CASE _inst_intStep OF
	0: // Reset FB and set default values
		IF NOT bModbusBusy AND NOT THIS^.P_bError THEN
			IF _in_bValue = TRUE THEN
				fbMBWriteSingleCoil.nValue := 16#FF00;
			ELSE
				fbMBWriteSingleCoil.nValue := 16#0000;
			END_IF
			fbMBWriteSingleCoil(
				sIPAddr:= in_sIPAddr, 
				nTCPPort:= in_uintTCPPort, 
				nUnitID:= in_byteUnitID, 
				nMBAddr:= _in_wordMBAddr, 
				bExecute:= FALSE, 
				tTimeout:= _in_timeTimeout);
		
			THIS^.M_LogMessage('Writing Single Coil');			
			_inst_intStep := 10;
		END_IF
		
		
	10: //Call ReadCoils Beckhoff Action and run it to completion
		fbMBWriteSingleCoil(bExecute := TRUE);
		IF NOT fbMBWriteSingleCoil.bBusy THEN
			fbMBWriteSingleCoil(bExecute:= FALSE);
			_inst_intStep := 20;
		END_IF
		
	20: //If no error, reset steps, else go to error step
		IF NOT fbMBWriteSingleCoil.bError THEN
			M_WriteSingleCoil := TRUE;
			THIS^.M_LogMessage('Write Single Coil Complete');
			_inst_intStep := 0;
		ELSE
			_inst_intStep := 100;
		END_IF
		
	100: //Error
		THIS^.M_SetError(fbMBWriteSingleCoil.nErrId,
							'Error occurred when writing single coil.');
		_inst_intStep := 0;
		
END_CASE
bModbusBusy := _inst_intStep > 0;
intWriteSingleCoilStep := _inst_intStep;
END_METHOD

(* Modbus Function Code 6 = Write Single Register *)
(* This function is used for writing an individual output register. 16 bit access is used. *)
METHOD M_WriteSingleRegister : BOOL
VAR_INPUT
	(* Modbus Data Address from which the data are read from the end device(slave) *)
	_in_wordMBAddr : WORD;
	(* Value to be written into the register (word value) *)
	_in_nValue : WORD;
	(* Timeout value for waiting for a response from the addressed slave *)
	_in_timeTimeout : TIME;
END_VAR
VAR_INST
	_inst_intStep: INT;
END_VAR
M_WriteSingleRegister := FALSE;

// Recover from premature stop
bWriteSingleRegisterBusy := TRUE;
_inst_intStep := intWriteSingleRegisterStep;

CASE _inst_intStep OF
	0: // Reset FB and set default values
		IF NOT bModbusBusy AND NOT THIS^.P_bError THEN
			fbMBWriteSingleReg(
				sIPAddr:= in_sIPAddr, 
				nTCPPort:= in_uintTCPPort, 
				nUnitID:= in_byteUnitID, 
				nMBAddr:= _in_wordMBAddr, 
				nValue:= _in_nValue, 
				bExecute:= FALSE, 
				tTimeout:= _in_timeTimeout);
		
			THIS^.M_LogMessage('Write Single Register');			
			_inst_intStep := 10;
		END_IF
		
		
	10: //Call ReadCoils Beckhoff Action and run it to completion
		fbMBWriteSingleReg(bExecute:= TRUE);
		IF NOT fbMBWriteSingleReg.bBusy THEN
			fbMBWriteSingleReg(bExecute:= FALSE);
			_inst_intStep := 20;
		END_IF
		
	20: //If no error, reset steps, else go to error step
		IF NOT fbMBWriteSingleReg.bError THEN
			M_WriteSingleRegister := TRUE;
			THIS^.M_LogMessage('Write Single Register Complete');
			_inst_intStep := 0;
		ELSE
			_inst_intStep := 100;
		END_IF
		
	100: //Error
		THIS^.M_SetError(fbMBWriteSingleReg.nErrId,
							'Error occurred when Writing Single Register.');
		_inst_intStep := 0;
		
END_CASE
bModbusBusy := _inst_intStep > 0;
intWriteSingleRegisterStep := _inst_intStep;
END_METHOD

(* This property should be TRUE while any method in this interface is actively
	executing, or FALSE otherwise. *)
PROPERTY P_bModbusBusy : BOOL
GET
P_bModbusBusy := bModbusBusy;
END_GET
END_PROPERTY

ACTION A_CommandRecovery:
// Methods have to explicitly set index busy as true each cycle
bModbusBusy := FALSE;

IF NOT bReadCoilsBusy AND intReadCoilsStep > 0 THEN
	intReadCoilsStep := 0;
	THIS^.M_LogWarning('M_ReadCoils stopped prematurely!');
END_IF
bReadCoilsBusy := FALSE;

IF NOT bReadInputRegsBusy AND intReadInputRegsStep > 0 THEN
	intReadInputRegsStep := 0;
	THIS^.M_LogWarning('M_ReadInputRegs stopped prematurely!');
END_IF
bReadInputRegsBusy := FALSE;

IF NOT bReadInputStatusBusy AND intReadInputStatusStep > 0 THEN
	intReadInputStatusStep := 0;
	THIS^.M_LogWarning('M_ReadInputStatus stopped prematurely!');
END_IF
bReadInputStatusBusy := FALSE;

IF NOT bReadRegsBusy AND intReadRegsStep > 0 THEN
	intReadRegsStep := 0;
	THIS^.M_LogWarning('M_ReadRegs stopped prematurely!');
END_IF
bReadRegsBusy := FALSE;

IF NOT bWriteMultipleCoilsBusy AND intWriteMultipleCoilsStep > 0 THEN
	intWriteMultipleCoilsStep := 0;
	THIS^.M_LogWarning('M_WriteMultipleCoils stopped prematurely!');
END_IF
bWriteMultipleCoilsBusy := FALSE;

IF NOT bWriteRegsBusy AND intWriteRegsStep > 0 THEN
	intWriteRegsStep := 0;
	THIS^.M_LogWarning('M_WriteRegs stopped prematurely!');
END_IF
bWriteRegsBusy := FALSE;

IF NOT bWriteSingleCoilBusy AND intWriteSingleCoilStep > 0 THEN
	intWriteSingleCoilStep := 0;
	THIS^.M_LogWarning('M_WriteSingleCoil stopped prematurely!');
END_IF
bWriteSingleCoilBusy := FALSE;

IF NOT bWriteSingleRegisterBusy AND intWriteSingleRegisterStep > 0 THEN
	intWriteSingleRegisterStep := 0;
	THIS^.M_LogWarning('M_WriteSingleRegister stopped prematurely!');
END_IF
bWriteSingleRegisterBusy := FALSE;
END_ACTION

END_FUNCTION_BLOCK

// Concrete/Resource Manager/FB_FifoBufferResMgr
(* FB to manage a shared resource. *)
FUNCTION_BLOCK FB_FifoBufferResMgr EXTENDS FB_ResourceManager IMPLEMENTS I_ResourceManagement, I_Resettable
VAR CONSTANT
	uintQUEUE_SIZE : UINT := 256;
END_VAR
VAR_INPUT
END_VAR
VAR_OUTPUT
END_VAR
VAR
	(* ID queue for checking out. *)
	arrQueue: ARRAY[1..uintQUEUE_SIZE] OF T_MaxString;
	strLastCheckout: STRING(255);
END_VAR

IF (strLastCheckout <> arrQueue[1]) AND LEN(arrQueue[1]) > 0 THEN
	M_LogMessage(CONCAT('Checked out by ', arrQueue[1]));
END_IF
strLastCheckout := arrQueue[1];

(* This should clear any errors on the device and bring it to a state where
	it is ready to be energized or otherwise activated. *)
METHOD M_Reset : BOOL
VAR
	arrBlankArray: ARRAY[1..uintQUEUE_SIZE] OF T_MaxString;
END_VAR
arrQueue := arrBlankArray;
M_Reset := TRUE;
END_METHOD

(* This property should be TRUE while any method in this interface is actively
	executing, or FALSE otherwise. *)
PROPERTY P_bResetBusy : BOOL
GET
P_bResetBusy := FALSE;
END_GET
END_PROPERTY

(* Checks in the resource for the given module. *)
METHOD M_CheckIn : BOOL
VAR_INPUT
	(* ID of the module checking the resource out. *)
	_in_strId	: Tc2_System.T_MaxString;
END_VAR
VAR
	_uintIndex: UINT;
	_bDeleted: BOOL;
	_uintStartIndex: UINT;
END_VAR
// Find and delete the given ID from the queue
_bDeleted := FALSE;
FOR _uintIndex := 1 TO uintQUEUE_SIZE DO
	IF LEN(arrQueue[_uintIndex]) <= 0 OR LEN(_in_strId) <= 0 THEN
		EXIT;
	ELSIF arrQueue[_uintIndex] = _in_strId THEN
		//THIS^.M_LogMessage(CONCAT('Checked in ', arrQueue[_uintIndex]));
		arrQueue[_uintIndex] := '';
		_bDeleted := TRUE;
		EXIT;
	END_IF
END_FOR

// If the ID was found and deleted, shift the other data to the left
IF _bDeleted AND _uintIndex < uintQUEUE_SIZE THEN
	_uintStartIndex := _uintIndex;
	FOR _uintIndex := _uintStartIndex TO (uintQUEUE_SIZE - 1) DO
		// If the next index is empty, assume rest of queue is empty
		IF LEN(arrQueue[_uintIndex+1]) <= 0 THEN
			EXIT;
		// Else shift the next index into the current index
		ELSE
			arrQueue[_uintIndex] := arrQueue[_uintIndex+1];
			arrQueue[_uintIndex+1] := '';
		END_IF
	END_FOR
END_IF

// Return TRUE
M_CheckIn := TRUE;
END_METHOD

(* Checks out the resource for the given module ID. *)
METHOD M_CheckOut : BOOL
VAR_INPUT
	(* ID of the module checking the resource out. *)
	_in_strId	: Tc2_System.T_MaxString;
END_VAR

VAR
	_uintIndex: UINT;
END_VAR
M_CheckOut := FALSE;

IF LEN(_in_strId) > 0 THEN
	// If the resource is checked out by the current ID, return TRUE
	IF arrQueue[1] = _in_strId THEN
		M_CheckOut := TRUE;
	// If the resource is not checked out at all, check it out
	ELSIF LEN(arrQueue[1]) <= 0 THEN
		arrQueue[1] := _in_strId;
		M_CheckOut := TRUE;
	// Else add the ID to the queue
	ELSE
		// Check that the ID is in the queue and add it if not
		FOR _uintIndex := 1 TO uintQUEUE_SIZE DO
			IF arrQueue[_uintIndex] = _in_strId THEN
				EXIT;
			ELSIF LEN(arrQueue[_uintIndex]) <= 0 THEN
				arrQueue[_uintIndex] := _in_strId;
				EXIT;
			END_IF
		END_FOR
	END_IF
END_IF
END_METHOD

(* TRUE if the resource is checked out. *)
PROPERTY P_bCheckedOut : BOOL
GET
P_bCheckedOut := LEN(arrQueue[1]) > 0;
END_GET
END_PROPERTY

(* ID of the module checking out the resource. *)
PROPERTY P_strCheckedOutBy : Tc2_System.T_MaxString
GET
P_strCheckedOutBy := arrQueue[1];
END_GET
END_PROPERTY

END_FUNCTION_BLOCK

// Functions/F_ButtonToggle
FUNCTION F_ButtonToggle : BOOL
VAR_INPUT
END_VAR
VAR_IN_OUT
	inout_bButton: BOOL;
	inout_bLastValue: BOOL;
END_VAR

IF inout_bButton THEN
	IF inout_bLastValue THEN
		inout_bButton := FALSE;
		inout_bLastValue := FALSE;
	ELSE
		inout_bLastValue := TRUE;
	END_IF
ELSE
	inout_bLastValue := FALSE;
END_IF

END_FUNCTION

// Functions/F_CalcCycleTime
FUNCTION F_CalcCycleTime : BOOL
VAR_INPUT
	in_timeStartTime: TIME;
END_VAR
VAR_OUTPUT
	out_timeEndTime: TIME;
	out_timeCycleTime: TIME;
END_VAR

out_timeEndTime := TIME();
out_timeCycleTime := out_timeEndTime - in_timeStartTime;
F_CalcCycleTime := TRUE;

END_FUNCTION

// Interfaces/Obsolete/I_ModularAPI
INTERFACE I_ModularAPI

(* Calls a method on the modular API, and returns true once
	the result of the method is received. *)
METHOD M_CallMethod : BOOL
VAR_INPUT
	(* ID of the module the method is being routed to. *)
	strModuleId: T_MaxString;
	
	(* Name of the API method that will be called. *)
	strMethodName: T_MaxString;
	
	(* An array of array of strings representing the name:value pair
		for all of the required method parameters. *)
	arrParameters: T_ApiMethodParameters;
END_VAR
VAR_OUTPUT
	(* Should be TRUE if the method executed without error. *)
	bSuccessful: BOOL;
	
	(* The return value of the method. *)
	strReturnValue: T_MaxString;
	
	(* Name:value pairs for any outputs of the method. *)
	arrOutputValues: T_ApiMethodParameters;
END_VAR
END_METHOD

(* Should return TRUE if there is a method in this interface that
	is executing. *)
PROPERTY P_bApiBusy : BOOL
GET
END_GET
END_PROPERTY

END_INTERFACE

// Project Information/F_GetCompany
// This function has been automatically generated from the project information.
{attribute 'signature_flag' := '1073741824'}
{attribute 'TcGenerated'}
{attribute 'no-analysis'}
FUNCTION F_GetCompany : WSTRING
VAR_INPUT
	
END_VAR

F_GetCompany := "Sensata Technologies";

END_FUNCTION

// Project Information/F_GetTitle
// This function has been automatically generated from the project information.
{attribute 'signature_flag' := '1073741824'}
{attribute 'TcGenerated'}
{attribute 'no-analysis'}
FUNCTION F_GetTitle : WSTRING
VAR_INPUT
	
END_VAR

F_GetTitle := "Sensata_Utilities";

END_FUNCTION

// Project Information/F_GetVersion
// This function has been automatically generated from the project information.
{attribute 'signature_flag' := '1073741824'}
{attribute 'TcGenerated'}
{attribute 'no-analysis'}
FUNCTION F_GetVersion : ST_LibVersion
VAR_INPUT
	
END_VAR

F_GetVersion.iMajor := 1;
F_GetVersion.iMinor := 0;
F_GetVersion.iBuild := 2;
F_GetVersion.iRevision := 0;
F_GetVersion.sVersion := '1.0.2';
F_GetVersion.nFlags := 0;

END_FUNCTION
